Universal Robots PolyScope program: URClient.urp

ProgramRoot directory=/home/ur/ursim-3.1/programs/URClient; kinematics=(a=[0, -0.425, -0.39225, 0, 0, 0], d=[0.08916, 0, 0, 0.10915, 0.09465, 0.0823], alpha=[1.5708, 0, 0, 1.5708, -1.5708, 0], deltaTheta=[0, 0, 0, 0, 0, 0], status=notInitialized); lastSavedInVersion=(project__name=Polyscope, major__version=3, minor__version=1, svn__revision=17195, build__date=Mar 11 2015, 13:02:28); name=URClient; programVersion=(project__name=Polyscope, major__version=3, minor__version=1, svn__revision=17195, build__date=Mar 11 2015, 13:02:28); robotEnvironmentFileName=default; serialNumberRobot=2014350001
  BeforeStart description=COMMAND_SEQUENCE_BEFORE_PROGRAM_START; name=BeforeStart
    Assignment expr=socket_open("127.0.0.1",21); operatorValueType=INTEGER; valueSource=EXPRESSION
    While count=0; expr=ExpressionVariableNode≟ False; type=LOOP_EXPR
      Assignment expr=socket_open("127.0.0.1",21); operatorValueType=INTEGER; valueSource=EXPRESSION
    Assignment expr=p[0,0,0,0,0,0]; operatorValueType=INTEGER; valueSource=EXPRESSION
    Assignment expr=6; operatorValueType=INTEGER; valueSource=EXPRESSION
  MainProgram cartesianAcceleration=1.2; cartesianSpeed=0.25; jointAcceleration=1.3962634015954636; jointSpeed=1.0471975511965976; sharedProcessMoveBlendRadius=0.025; motionType=JOINT_SPACE
    Assignment assignmentOperatorMessage=send to server; operatorValueType=STRING; valueSource=OPERATOR
    Script type=0; expressionBranchNode=socket_send_string(ExpressionVariableNode)
    Assignment expr=socket_read_ascii_float(6); operatorValueType=INTEGER; valueSource=EXPRESSION
    While count=0; expr=ExpressionVariableNode[0]≠6; type=LOOP_EXPR
      Wait 
      Assignment expr=socket_read_ascii_float(6); operatorValueType=INTEGER; valueSource=EXPRESSION
    While count=0; expr=ExpressionVariableNode<6; type=LOOP_EXPR
      Script type=0; expressionBranchNode=ExpressionVariableNode[ExpressionVariableNode]=ExpressionVariableNode[ExpressionVariableNode+1]
      Assignment expr=ExpressionVariableNode+1; operatorValueType=INTEGER; valueSource=EXPRESSION
    Move cartesianAcceleration=1.2; cartesianSpeed=0.25; jointAcceleration=1.3962634015954636; jointSpeed=1.0471975511965976; sharedProcessMoveBlendRadius=0.025; motionType=JOINT_SPACE
      Waypoint blendRadius=0.05; cartesianAcceleration=1.2; cartesianSpeed=0.25; jointAcceleration=1.3962634015954636; jointSpeed=1.0471975511965976; nextMotionTime=2.0; stoppoint=true; useSharedBlendParameter=true; useSharedParameters=true; positionType=VARIABLE_POSITION; name=Waypoint
